FUNCTION_BLOCK E_SPLIT2
  (* Version 1.0, 2005-06-12, Goran Cengic, Chalmers *)
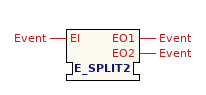
  EVENT_INPUT
    EI;
  END_EVENT
  EVENT_OUTPUT
    EO1;
    EO2;
  END_EVENT
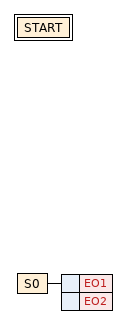
  EC_STATES
    START;
    S0 : -> EO1, -> EO2;
  END_STATES
  EC_TRANSITIONS
    START TO SO := EI;
    SO TO START := 1;
  END_TRANSITIONS
END_FUNCTION_BLOCK
